# EPICS StreamDevice protocol: streamDevice/rosie.proto
# DolphinDAQ Rosie protocol file
# Built by examining examples at: https://paulscherrerinstitute.github.io/StreamDevice/protocol.html#gen
# And also by examining input/output formats at https://paulscherrerinstitute.github.io/StreamDevice/formats.html

Terminator = CR LF;

##### Common #####

info {
	ExtraInput = Ignore;
	out "*IDN?";
	in "%39c";
}

debug {
   ExtraInput = Ignore;
   out "%s";
   in "%39c";
}

CountQ {
        out ":TRIGger:COUNt?";
        in "%u";
    }

Count {
        out ":TRIGger:COUNt %u";
        @init { CountQ; }
    }

DecimationQ {
        out ":TRIGger:DECimation?";
        in "%u";
    }

Decimation {
        out ":TRIGger:DECimation %u";
        @init { DecimationQ; }
    }

TimeQ {
        out ":SYSTem:TIME?";
	    in "%39c";
    }

TimeUnixQ {
        out ":SYSTem:TIME:UNIX?";
        in "%i";
    }

TimeUnix {
        out ":SYSTem:TIME:UNIX %i";
        @init { TimeUnixQ; }
    }

##### Rosie-Specific #####

OutEnabledQ {
        out ":ROSie:OUTPut:ENabled?";
        in "%i";
    }

OutEnabled {
        out ":ROSie:OUTPut:ENabled %i";
        @init { OutEnabledQ; }
    }

OutFirstQ {
        out ":ROSie:OUTPut:FIRSt?";
        in "%u";
    }

OutCountQ {
        out ":ROSie:OUTPut:COUNt?";
        in "%u";
    }
